(* PLC project io_engine_2d1s, Dassault Systèmes ControlBuild 2024x *)
(* stored: creationDateTime 2023-10-03T11:12:46-01:00 *)

PROGRAM panel
  VAR_OUTPUT
    forwardPB : BOOL := false;
    backwardPB : BOOL := false;
    stopPB : BOOL := false;
  END_VAR

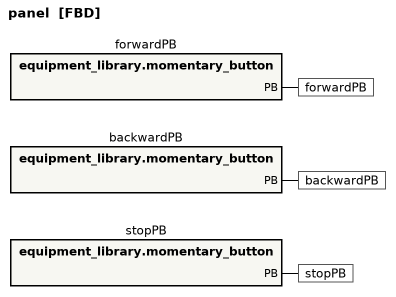
(* FBD diagram, written out as Structured Text *)
forwardPB();
forwardPB := forwardPB.PB;
backwardPB();
backwardPB := backwardPB.PB;
stopPB();
stopPB := stopPB.PB;
END_PROGRAM

(* Integrated object C/C+OP of a motor with one speed and two directions *)
PROGRAM io_library.io_engine_2d1s
  VAR_INPUT
    autoMode : BOOL := false;
    manualMode : BOOL := false;
  END_VAR
  VAR_INPUT
    autoFwdCmd : BOOL := false;
    autoBwdCmd : BOOL := false;
  END_VAR
  VAR_INPUT
    acknowledgePB : BOOL := false;
  END_VAR
  VAR_OUTPUT
    speedVal : REAL := 0.0;
    speedPercent : REAL := 0.0;
  END_VAR
  VAR_OUTPUT
    generalFault : BOOL := false;
  END_VAR

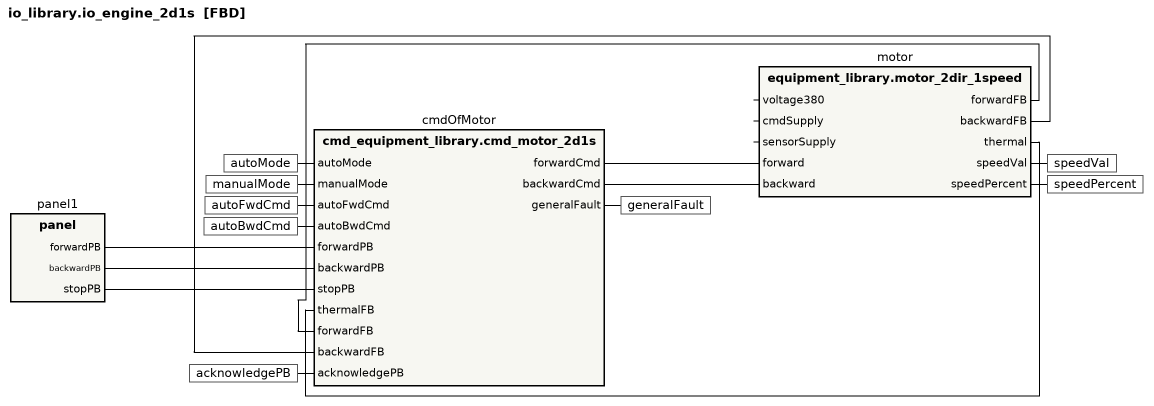
(* FBD diagram, written out as Structured Text *)
panel1();
motor(forward := cmdOfMotor.forwardCmd, backward := cmdOfMotor.backwardCmd);
cmdOfMotor(autoMode := autoMode, manualMode := manualMode, autoFwdCmd := autoFwdCmd, autoBwdCmd := autoBwdCmd, forwardPB := panel1.forwardPB, backwardPB := panel1.backwardPB, stopPB := panel1.stopPB, thermalFB := motor.thermal, forwardFB := motor.forwardFB, backwardFB := motor.backwardFB, acknowledgePB := acknowledgePB);
generalFault := cmdOfMotor.generalFault;
speedVal := motor.speedVal;
speedPercent := motor.speedPercent;
END_PROGRAM
